	(* Get the direction of the local x-axis. *)
	METHOD GetDirectionX
	VAR_IN_OUT
		(* The local x-direction of this orientation. *)
 {attribute 'GUID' := '26B8CE0C-6327-CF56-46C9-563EF634067D'}
				localX : TangentXY;
	END_VAR
END_METHOD


	(* Get the direction of the local y-axis. *)
	METHOD GetDirectionY
	VAR_IN_OUT
		(* The local y-direction of this orientation. *)
 {attribute 'GUID' := '26B8CE0C-6327-CF56-46C9-563EF634067D'}
				localY : TangentXY;
	END_VAR
END_METHOD


	(* Invert this position. *)
	METHOD Invert
END_METHOD


	(* Multiply an orientation to this orientation. *)
	METHOD ConcatenateWith
	VAR_IN_OUT
		(* Orientation to concatenate with. *)
 {attribute 'GUID' := 'ECEACC25-61F8-C229-5DF2-DD8132935CEE'}
				orientation2D : Orientation2D;
	END_VAR
END_METHOD


	(* Turn the orientation. *)
	METHOD TurnByC
	VAR_INPUT
		(* Rotation angle to turn by in degrees [°]. *)
		angle : LREAL;
	END_VAR
END_METHOD


	(* Rotate a PositionXY according to this orientation. *)
	METHOD Transform
	VAR_IN_OUT
		(* The orientation to multipy by. *)
 {attribute 'GUID' := '96F2C7F9-077A-C570-41B3-040B08209702'}
				positionXY : PositionXY;
	END_VAR
END_METHOD


	PROPERTY angle : LREAL
SET
END_SET
GET
END_GET
END_PROPERTY

END_FUNCTION_BLOCK

// POUs/Spatial/Functions/ConcatenateABC

	{attribute 'TcIecLibraryType'}
	{attribute 'external_name' := 'ConcatenateABC_GUID_186C30DE_4777_CF4B_4981_F8D310866484'}
	(* Concatenate two instances of Orientation3D. *)
	FUNCTION ConcatenateABC : BOOL
	VAR_IN_OUT
		rotation0	:	Orientation3D;	(* 1st input orientation of the concatenation. *)
		rotation1	:	Orientation3D;	(* 2nd input orientation of the concatenation. *)
		concatenation	:	Orientation3D;	(* The concatenation of the two input instances. *)
	END_VAR

END_FUNCTION

// POUs/Spatial/Positions/Orientation3D

	{attribute 'c++_compatible'}
	{attribute 'external_name' := 'Orientation3D_GUID_88260D10_4258_CB4B_4E9C_4A364CDA3C22'}
	{attribute 'TcIecLibraryType'}
	{attribute 'no_explicit_call' :='do not call this POU directly'}
	{attribute 'no_assign'}
	(* 3D orientation. All angles in degrees [°]. *)
	FUNCTION_BLOCK Orientation3D
	VAR
		(* Rotation around the 1st local axis in degrees [°]. *)
		p0 : LREAL;
		(* Rotation around 2nd local axis in degrees [°]. *)
		p1 : LREAL;
		(* Rotation around 3rd local axis in degrees [°]. *)
		p2 : LREAL;
		(* Defines the rotation order (rotate around local axes from left to right) *)
		 {attribute 'GUID' := 'BF8BCC1E-925E-4A57-801C-CC42AFDDA86D'}
		coordinates : E_RotationCoordinates := E_RotationCoordinates.CBA;
		 {attribute 'hide'}
		_reserved1 : ARRAY [1..84] OF USINT;
	END_VAR


	(* Internal method *)
	{attribute 'hide'}
	METHOD FB_init : BOOL
	VAR_INPUT
		(*  if TRUE, the retain variables are initialized (warm start / cold start) *)
		bInitRetains : BOOL;
		(*  if TRUE, the instance afterwards gets moved into the copy code (online change) *)
		bInCopyCode : BOOL;
	END_VAR
END_METHOD


	(* Internal method *)
	{attribute 'hide'}
	METHOD FB_exit : BOOL
	VAR_INPUT
		(*  if TRUE, the exit method is called for exiting an instance that is copied afterwards (online change). *)
		bInCopyCode : BOOL;
	END_VAR
END_METHOD


	(* Set the components of this vector to '0.0'. *)
	METHOD SetZero
END_METHOD


	(* Set the components of this position. *)
	METHOD SetValues
	VAR_IN_OUT
		(* The position values to set. *)
 {attribute 'GUID' := '88260D10-4258-CB4B-4E9C-4A364CDA3C22'}
				orientation3D : Orientation3D;
	END_VAR
END_METHOD


	(* Set the coordinates of the orientation. *)
	METHOD SetValuesABC
	VAR_INPUT
		(* 1st rotation angle in degrees [°]. *)
		phi0 : LREAL;
		(* 2nd rotation angle in degrees [°]. *)
		phi1 : LREAL;
		(* 3rd rotation angle in degrees [°]. *)
		phi2 : LREAL;
	END_VAR
END_METHOD


	(* Set the coordinates of the orientation. *)
	METHOD SetValuesACB
	VAR_INPUT
		(* 1st rotation angle in degrees [°]. *)
		phi0 : LREAL;
		(* 2nd rotation angle in degrees [°]. *)
		phi1 : LREAL;
		(* 3rd rotation angle in degrees [°]. *)
		phi2 : LREAL;
	END_VAR
END_METHOD


	(* Set the coordinates of the orientation. *)
	METHOD SetValuesBCA
	VAR_INPUT
		(* 1st rotation angle in degrees [°]. *)
		phi0 : LREAL;
		(* 2nd rotation angle in degrees [°]. *)
		phi1 : LREAL;
		(* 3rd rotation angle in degrees [°]. *)
		phi2 : LREAL;
	END_VAR
END_METHOD


	(* Set the coordinates of the orientation. *)
	METHOD SetValuesBAC
	VAR_INPUT
		(* 1st rotation angle in degrees [°]. *)
		phi0 : LREAL;
		(* 2nd rotation angle in degrees [°]. *)
		phi1 : LREAL;
		(* 3rd rotation angle in degrees [°]. *)
		phi2 : LREAL;
	END_VAR
END_METHOD


	(* Set the coordinates of the orientation. *)
	METHOD SetValuesCAB
	VAR_INPUT
		(* 1st rotation angle in degrees [°]. *)
		phi0 : LREAL;
		(* 2nd rotation angle in degrees [°]. *)
		phi1 : LREAL;
		(* 3rd rotation angle in degrees [°]. *)
		phi2 : LREAL;
	END_VAR
END_METHOD


	(* Set the coordinates of the orientation. *)
	METHOD SetValuesCBA
	VAR_INPUT
		(* 1st rotation angle in degrees [°]. *)
		phi0 : LREAL;
		(* 2nd rotation angle in degrees [°]. *)
		phi1 : LREAL;
		(* 3rd rotation angle in degrees [°]. *)
		phi2 : LREAL;
	END_VAR
END_METHOD


	(* Set the coordinates of the orientation. *)
	METHOD SetValuesABA
	VAR_INPUT
		(* 1st rotation angle in degrees [°]. *)
		phi0 : LREAL;
		(* 2nd rotation angle in degrees [°]. *)
		phi1 : LREAL;
		(* 3rd rotation angle in degrees [°]. *)
		phi2 : LREAL;
	END_VAR
END_METHOD


	(* Set the coordinates of the orientation. *)
	METHOD SetValuesACA
	VAR_INPUT
		(* 1st rotation angle in degrees [°]. *)
		phi0 : LREAL;
		(* 2nd rotation angle in degrees [°]. *)
		phi1 : LREAL;
		(* 3rd rotation angle in degrees [°]. *)
		phi2 : LREAL;
	END_VAR
END_METHOD


	(* Set the coordinates of the orientation. *)
	METHOD SetValuesBCB
	VAR_INPUT
		(* 1st rotation angle in degrees [°]. *)
		phi0 : LREAL;
		(* 2nd rotation angle in degrees [°]. *)
		phi1 : LREAL;
		(* 3rd rotation angle in degrees [°]. *)
		phi2 : LREAL;
	END_VAR
END_METHOD


	(* Set the coordinates of the orientation. *)
	METHOD SetValuesBAB
	VAR_INPUT
		(* 1st rotation angle in degrees [°]. *)
		phi0 : LREAL;
		(* 2nd rotation angle in degrees [°]. *)
		phi1 : LREAL;
		(* 3rd rotation angle in degrees [°]. *)
		phi2 : LREAL;
	END_VAR
END_METHOD


	(* Set the coordinates of the orientation. *)
	METHOD SetValuesCAC
	VAR_INPUT
		(* 1st rotation angle in degrees [°]. *)
		phi0 : LREAL;
		(* 2nd rotation angle in degrees [°]. *)
		phi1 : LREAL;
		(* 3rd rotation angle in degrees [°]. *)
		phi2 : LREAL;
	END_VAR
END_METHOD


	(* Set the coordinates of the orientation. *)
	METHOD SetValuesCBC
	VAR_INPUT
		(* 1st rotation angle in degrees [°]. *)
		phi0 : LREAL;
		(* 2nd rotation angle in degrees [°]. *)
		phi1 : LREAL;
		(* 3rd rotation angle in degrees [°]. *)
		phi2 : LREAL;
	END_VAR
END_METHOD


	(* Get the direction of the local x-axis. *)
	METHOD GetDirectionX
	VAR_IN_OUT
		(* The local x-direction of this orientation. *)
 {attribute 'GUID' := 'F5C610D1-97C6-C19E-7CED-E3534BCC46DA'}
				localX : Tangent3D;
	END_VAR
END_METHOD


	(* Get the direction of the local y-axis. *)
	METHOD GetDirectionY
	VAR_IN_OUT
		(* The local y-direction of this orientation. *)
 {attribute 'GUID' := 'F5C610D1-97C6-C19E-7CED-E3534BCC46DA'}
				localY : Tangent3D;
	END_VAR
END_METHOD


	(* Get the direction of the local z-axis. *)
	METHOD GetDirectionZ
	VAR_IN_OUT
		(* The local z-direction of this orientation. *)
 {attribute 'GUID' := 'F5C610D1-97C6-C19E-7CED-E3534BCC46DA'}
				localZ : Tangent3D;
	END_VAR
END_METHOD


	(* Invert this position. *)
	METHOD Invert
END_METHOD


	(* Multiply an orientation to this orientation. *)
	METHOD ConcatenateWith
	VAR_IN_OUT
		(* Orientation to concatenate with. *)
 {attribute 'GUID' := '88260D10-4258-CB4B-4E9C-4A364CDA3C22'}
				orientation : Orientation3D;
	END_VAR
END_METHOD


	(* Rotate around an arbitrary local axis. The turn angle is given by the length of the axis. *)
	METHOD TurnBy
	VAR_IN_OUT
		(* The axis of rotation. Its length represents the angle of rotation in degrees [°]. *)
 {attribute 'GUID' := '079EE0EF-BB9A-C328-4691-0C1D9775AB9B'}
				axis : TangentABC;
	END_VAR
END_METHOD


	(* Rotation around the local x-axis. *)
	METHOD TurnByA
	VAR_INPUT
		(* The angle to rotate by in degrees [°]. *)
		da : LREAL;
	END_VAR
END_METHOD


	(* Rotation around the local y-axis. *)
	METHOD TurnByB
	VAR_INPUT
		(* The angle to rotate by in degrees [°]. *)
		db : LREAL;
	END_VAR
END_METHOD


	(* Rotation around the local z-axis. *)
	METHOD TurnByC
	VAR_INPUT
		(* The angle to rotate by in degrees [°]. *)
		dc : LREAL;
	END_VAR
END_METHOD


	(* Rotate a Position3D according to this orientation. *)
	METHOD Transform
	VAR_IN_OUT
		(* Position to transform. *)
 {attribute 'GUID' := '2AB870EB-68E4-CB90-6B70-58195CE52F48'}
				position3D : Position3D;
	END_VAR
END_METHOD


	PROPERTY phi0 : LREAL
SET
END_SET
GET
END_GET
END_PROPERTY


	PROPERTY phi1 : LREAL
SET
END_SET
GET
END_GET
END_PROPERTY


	PROPERTY phi2 : LREAL
SET
END_SET
GET
END_GET
END_PROPERTY


	PROPERTY convention : E_RotationCoordinates
SET
END_SET
GET
END_GET
END_PROPERTY

END_FUNCTION_BLOCK

// POUs/Spatial/Functions/ConcatenateXYC

	{attribute 'TcIecLibraryType'}
	{attribute 'external_name' := 'ConcatenateXYC_GUID_3FF36687_1D56_CFED_49BA_E16821D33A61'}
	(* Concatenate two instances of PositionXYC. *)
	FUNCTION ConcatenateXYC : BOOL
	VAR_IN_OUT
		position0	:	PositionXYC;	(* 1st input position of the concatenation. *)
		position1	:	PositionXYC;	(* 2nd input position of the concatenation. *)
		concatenation	:	PositionXYC;	(* The concatenation of the two input instances. *)
	END_VAR

END_FUNCTION

// POUs/Spatial/Functions/AddXY

	{attribute 'TcIecLibraryType'}
	{attribute 'external_name' := 'AddXY_GUID_9AF6CBF8_E886_C1CE_7D79_B6347AC56EDE'}
	(* Add two instances of TangentXY. *)
	FUNCTION AddXY : BOOL
	VAR_IN_OUT
		tangent0	:	TangentXY;	(* 1st input tangent vector. *)
		tangent1	:	TangentXY;	(* 2nd input tangent vector. *)
		sumTangent	:	TangentXY;	(* Sum of the two tangent vectors. *)
	END_VAR

END_FUNCTION

// POUs/Spatial/Functions/SubtractXY

	{attribute 'TcIecLibraryType'}
	{attribute 'external_name' := 'SubtractXY_GUID_4B4AC809_E392_C314_4C45_4DF45CDC0C29'}
	(* Subtract two instances of TangentXY. *)
	FUNCTION SubtractXY : BOOL
	VAR_IN_OUT
		tangent0	:	TangentXY;	(* 1st input tangent vector. *)
		tangent1	:	TangentXY;	(* 2nd input tangent vector. *)
		difference	:	TangentXY;	(* Difference of the two tangent vectors. *)
	END_VAR

END_FUNCTION

// POUs/Spatial/Functions/MultiplyXY

	{attribute 'TcIecLibraryType'}
	{attribute 'external_name' := 'MultiplyXY_GUID_85E13E1D_F467_C3B1_4BCC_CCAD43989479'}
	(* Multiply a TangentXY by a scalar and return the result. *)
	FUNCTION MultiplyXY : BOOL
	VAR_IN_OUT
		tangent	:	TangentXY;	(* Tangent vector to multiply. *)
	END_VAR
	VAR_INPUT
		scalar	:	LREAL;	(* Scalar value to multiply with. *)
	END_VAR
	VAR_IN_OUT
		scaled	:	TangentXY;	(* Scaled input tangent vector. *)
	END_VAR

END_FUNCTION

// POUs/Spatial/Functions/ScalarXY

	{attribute 'TcIecLibraryType'}
	{attribute 'external_name' := 'ScalarXY_GUID_93FCFE61_1A57_C568_4366_FB966945F7BE'}
	(* Compute the scalar product of two instance of TangentXY. *)
	FUNCTION ScalarXY : LREAL
	VAR_IN_OUT
		tangent0	:	TangentXY;	(* 1st input tangent vector. *)
		tangent1	:	TangentXY;	(* 2nd input tangent vector. *)
	END_VAR

END_FUNCTION

// POUs/Spatial/Functions/Add3D

	{attribute 'TcIecLibraryType'}
	{attribute 'external_name' := 'Add3D_GUID_59367F1B_539F_CD33_6456_DF2799B8BB05'}
	(* Add two instances of Tangent3D. *)
	FUNCTION Add3D : BOOL
	VAR_IN_OUT
		tangent0	:	Tangent3D;	(* 1st input tangent vector. *)
		tangent1	:	Tangent3D;	(* 2nd input tangent vector. *)
		sumTangent	:	Tangent3D;	(* Sum of the two tangent vectors. *)
	END_VAR

END_FUNCTION

// POUs/Spatial/Functions/Subtract3D

	{attribute 'TcIecLibraryType'}
	{attribute 'external_name' := 'Subtract3D_GUID_4490D74F_E885_C89D_4A9C_8B24E18A51D7'}
	(* Subtract two instances of Tangent3D. *)
	FUNCTION Subtract3D : BOOL
	VAR_IN_OUT
		tangent0	:	Tangent3D;	(* 1st input tangent vector. *)
		tangent1	:	Tangent3D;	(* 2nd input tangent vector. *)
		difference	:	Tangent3D;	(* Difference of the two tangent vectors. *)
	END_VAR

END_FUNCTION

// POUs/Spatial/Functions/Multiply3D

	{attribute 'TcIecLibraryType'}
	{attribute 'external_name' := 'Multiply3D_GUID_383573DC_E2EF_CCC1_44E2_29017F46A5D5'}
	(* Multiply a Tangent3D by a scalar. *)
	FUNCTION Multiply3D : BOOL
	VAR_IN_OUT
		tangent	:	Tangent3D;	(* Tangent vector to multiply. *)
	END_VAR
	VAR_INPUT
		scalar	:	LREAL;	(* Scalar value to multiply with. *)
	END_VAR
	VAR_IN_OUT
		scaled	:	Tangent3D;	(* Scaled input tangent vector. *)
	END_VAR

END_FUNCTION

// POUs/Spatial/Functions/Scalar3D

	{attribute 'TcIecLibraryType'}
	{attribute 'external_name' := 'Scalar3D_GUID_CDD5D329_BF8D_CFD8_59AB_AE11960F9E3D'}
	(* Compute the scalar product of two instances of Tangent3D. *)
	FUNCTION Scalar3D : LREAL
	VAR_IN_OUT
		tangent0	:	Tangent3D;	(* 1st input tangent vector. *)
		tangent1	:	Tangent3D;	(* 2nd input tangent vector. *)
	END_VAR

END_FUNCTION

// POUs/Spatial/Functions/Cross3D

	{attribute 'TcIecLibraryType'}
	{attribute 'external_name' := 'Cross3D_GUID_18FD21AE_F556_CC15_6188_E6099864EA00'}
	(* Compute the cross product of two instances of Tangent3D. *)
	FUNCTION Cross3D : BOOL
	VAR_IN_OUT
		tangent0	:	Tangent3D;	(* 1st input tangent vector. *)
		tangent1	:	Tangent3D;	(* 2nd input tangent vector. *)
		crossProduct	:	Tangent3D;	(* The resulting cross product. *)
	END_VAR

END_FUNCTION

// POUs/Spatial/Functions/AddABC

	{attribute 'TcIecLibraryType'}
	{attribute 'external_name' := 'AddABC_GUID_C8FBE575_5501_C20B_7B10_541D2B8D8FAB'}
	(* Add two instances of TangentABC. *)
	FUNCTION AddABC : BOOL
	VAR_IN_OUT
		tangent0	:	TangentABC;	(* 1st input tangent vector. *)
		tangent1	:	TangentABC;	(* 2nd input tangent vector. *)
		sumTangent	:	TangentABC;	(* Sum of the two tangent vectors. *)
	END_VAR

END_FUNCTION

// POUs/Spatial/Functions/SubtractABC

	{attribute 'TcIecLibraryType'}
	{attribute 'external_name' := 'SubtractABC_GUID_75447D74_7EE7_C0D8_4EE5_65C72445BC2E'}
	(* Subtract two instances of TangentABC. *)
	FUNCTION SubtractABC : BOOL
	VAR_IN_OUT
		tangent0	:	TangentABC;	(* 1st input tangent vector. *)
		tangent1	:	TangentABC;	(* 2nd input tangent vector. *)
		difference	:	TangentABC;	(* Difference of the two tangent vectors. *)
	END_VAR

END_FUNCTION

// POUs/Spatial/Functions/MultiplyABC

	{attribute 'TcIecLibraryType'}
	{attribute 'external_name' := 'MultiplyABC_GUID_B5567C7B_8039_CF9D_597F_679077B14500'}
	(* Multiply a TangentABC by a scalar. *)
	FUNCTION MultiplyABC : BOOL
	VAR_IN_OUT
		tangent	:	TangentABC;	(* Tangent vector to multiply. *)
	END_VAR
	VAR_INPUT
		scalar	:	LREAL;	(* Scalar value to multiply with. *)
	END_VAR
	VAR_IN_OUT
		scaled	:	TangentABC;	(* Scaled input tangent vector. *)
	END_VAR

END_FUNCTION

// POUs/Spatial/Functions/AddXYC

	{attribute 'TcIecLibraryType'}
	{attribute 'external_name' := 'AddXYC_GUID_6597480E_11BA_C407_44FC_28CB30711289'}
	(* Add two instances of TangentXYC. *)
	FUNCTION AddXYC : BOOL
	VAR_IN_OUT
		tangent0	:	TangentXYC;	(* 1st input tangent vector. *)
		tangent1	:	TangentXYC;	(* 2nd input tangent vector. *)
		sumTangent	:	TangentXYC;	(* Sum of the two tangent vectors. *)
	END_VAR

END_FUNCTION

// POUs/Spatial/Functions/SubtractXYC

	{attribute 'TcIecLibraryType'}
	{attribute 'external_name' := 'SubtractXYC_GUID_A66A1E91_4274_CA5D_7BE9_ABF8824078CE'}
	(* Subtract two instances of TangentXYC. *)
	FUNCTION SubtractXYC : BOOL
	VAR_IN_OUT
		tangent0	:	TangentXYC;	(* 1st input tangent vector. *)
		tangent1	:	TangentXYC;	(* 2nd input tangent vector. *)
		difference	:	TangentXYC;	(* Difference of the two tangent vectors. *)
	END_VAR

END_FUNCTION

// POUs/Spatial/Functions/MultiplyXYC

	{attribute 'TcIecLibraryType'}
	{attribute 'external_name' := 'MultiplyXYC_GUID_10B08A83_42B7_C12E_7EDD_506DEB6C7E94'}
	(* Multiply a TangentXYC by a scalar. *)
	FUNCTION MultiplyXYC : BOOL
	VAR_IN_OUT
		tangent	:	TangentXYC;	(* Tangent vector to multiply. *)
	END_VAR
	VAR_INPUT
		scalar	:	LREAL;	(* Scalar value to multiply with. *)
	END_VAR
	VAR_IN_OUT
		scaled	:	TangentXYC;	(* Scaled input tangent vector. *)
	END_VAR

END_FUNCTION

// POUs/Spatial/Functions/Add6D

	{attribute 'TcIecLibraryType'}
	{attribute 'external_name' := 'Add6D_GUID_70971E3D_141C_C82B_491A_28750F021F76'}
	(* Add two instances of Tangent6D. *)
	FUNCTION Add6D : BOOL
	VAR_IN_OUT
		tangent0	:	Tangent6D;	(* 1st input tangent vector. *)
		tangent1	:	Tangent6D;	(* 2nd input tangent vector. *)
		sumTangent	:	Tangent6D;	(* Sum of the two tangent vectors. *)
	END_VAR

END_FUNCTION

// POUs/Spatial/Functions/Subtract6D

	{attribute 'TcIecLibraryType'}
	{attribute 'external_name' := 'Subtract6D_GUID_850464F7_0919_C7C4_6C69_D5D4CC7F433D'}
	(* Subtract two instances of Tangent6D. *)
	FUNCTION Subtract6D : BOOL
	VAR_IN_OUT
		tangent0	:	Tangent6D;	(* 1st input tangent vector. *)
		tangent1	:	Tangent6D;	(* 2nd input tangent vector. *)
		difference	:	Tangent6D;	(* Difference of the two tangent vectors. *)
	END_VAR

END_FUNCTION

// POUs/Spatial/Functions/Multiply6D

	{attribute 'TcIecLibraryType'}
	{attribute 'external_name' := 'Multiply6D_GUID_91590C66_6BA7_C429_76E4_214A1B0FF139'}
	(* Multiply a Tangent6D by a scalar. *)
	FUNCTION Multiply6D : BOOL
	VAR_IN_OUT
		tangent	:	Tangent6D;	(* Tangent vector to multiply. *)
	END_VAR
	VAR_INPUT
		scalar	:	LREAL;	(* Scalar value to multiply with. *)
	END_VAR
	VAR_IN_OUT
		scaled	:	Tangent6D;	(* Scaled input tangent vector. *)
	END_VAR

END_FUNCTION

// POUs/Spatial/Functions/ConvertToCartesian2D

	{attribute 'TcIecLibraryType'}
	{attribute 'external_name' := 'ConvertToCartesian2D_GUID_1DE05828_63AC_CD5B_493C_397BF5B8F2DA'}
	(* Convert local XYC-dynamic properties to global XY ones. *)
	FUNCTION ConvertToCartesian2D : BOOL
	VAR_IN_OUT
		position	:	PositionXYC;	(* The position hosting the local dynamic state. *)
		velocity	:	TangentXYC;	(* The local velocity vector. *)
		acceleration	:	TangentXYC;	(* The local acceleration vector. *)
		velocity_XY	:	TangentXY;	(* The resulting global Cartesian velocity. *)
		acceleration_XY	:	TangentXY;	(* The resulting global Cartesian acceleration. *)
	END_VAR

END_FUNCTION

// POUs/Shapes/Geometry2D/Container2D

	{attribute 'c++_compatible'}
	{attribute 'external_name' := 'Container2D_GUID_315B01A2_C609_C244_71C6_4F8CF4BA2CAC'}
	{attribute 'TcIecLibraryType'}
	{attribute 'no_explicit_call' :='do not call this POU directly'}
	{attribute 'no_assign'}
	FUNCTION_BLOCK Container2D EXTENDS Geometry2D


	(* Internal method *)
	METHOD FB_init : BOOL
	VAR_INPUT
		(*  if TRUE, the retain variables are initialized (warm start / cold start) *)
		bInitRetains : BOOL;
		(*  if TRUE, the instance afterwards gets moved into the copy code (online change) *)
		bInCopyCode : BOOL;
	END_VAR
END_METHOD


	(* Internal method *)
	{attribute 'hide'}
	METHOD FB_exit : BOOL
	VAR_INPUT
		(*  if TRUE, the exit method is called for exiting an instance that is copied afterwards (online change). *)
		bInCopyCode : BOOL;
	END_VAR
END_METHOD


	(* Add a geometry to the container. *)
	METHOD AddElement : UDINT
	VAR_IN_OUT
		(* The geometry to add. *)
 {attribute 'GUID' := 'AD3CB6DF-15CC-CB02-52B0-F7F4EE14B341'}
				inputObject : Geometry2D;
	END_VAR
END_METHOD


	(* Remove a specified geometry from the container. *)
	METHOD RemoveElement
	VAR_INPUT
		(* ID of the geometry to remove. *)
		id : UDINT;
	END_VAR
END_METHOD


	(* Remove all geometries from the container. *)
	METHOD Clear
END_METHOD


	(* Get the number of geometry elements in container. *)
	METHOD GetCount : UDINT
END_METHOD


	(* Get the combined boundary of all hosted 2D-geometries. *)
	METHOD GetBoundary
	VAR_IN_OUT
		(* The combined boundary.. *)
 {attribute 'GUID' := '315B01A2-C609-C244-71C6-4F8CF4BA2CAC'}
				boundary : Container2D;
	END_VAR
END_METHOD

END_FUNCTION_BLOCK

// POUs/Shapes/Geometry2D/Extrude2D

	{attribute 'c++_compatible'}
	{attribute 'external_name' := 'Extrude2D_GUID_A7398709_3D7C_C1FD_7FCC_D371605A7865'}
	{attribute 'TcIecLibraryType'}
	{attribute 'no_explicit_call' :='do not call this POU directly'}
	{attribute 'no_assign'}
	FUNCTION_BLOCK Extrude2D EXTENDS Geometry2D


	(* Internal method *)
	METHOD FB_init : BOOL
	VAR_INPUT
		(*  if TRUE, the retain variables are initialized (warm start / cold start) *)
		bInitRetains : BOOL;
		(*  if TRUE, the instance afterwards gets moved into the copy code (online change) *)
		bInCopyCode : BOOL;
	END_VAR
END_METHOD


	(* Internal method *)
	{attribute 'hide'}
	METHOD FB_exit : BOOL
	VAR_INPUT
		(*  if TRUE, the exit method is called for exiting an instance that is copied afterwards (online change). *)
		bInCopyCode : BOOL;
	END_VAR
END_METHOD


	(* Define the extrusion geometry by a path and the corners to extrude. *)
	METHOD ExtrudeAlong
	VAR_IN_OUT
		(* The path to extrude along. *)
 {attribute 'GUID' := '044C9999-A9FC-C11F-572C-C4386A916232'}
				path : PathXYC;
	END_VAR
	VAR_INPUT
		(* 1st distance from the path to extrude. *)
		dy0 : LREAL;
		(* 2nd distance from the path to extrude. *)
		dy1 : LREAL;
		(* Number of steps to employ along the path. *)
		extrusionSteps : UDINT;
	END_VAR
END_METHOD


	(* Check whether this extrusion geometry is valid. *)
	METHOD IsValid : BOOL
END_METHOD

END_FUNCTION_BLOCK

// POUs/Paths/Components/PathXYC

	{attribute 'c++_compatible'}
	{attribute 'external_name' := 'PathXYC_GUID_044C9999_A9FC_C11F_572C_C4386A916232'}
	{attribute 'TcIecLibraryType'}
	{attribute 'no_explicit_call' :='do not call this POU directly'}
	{attribute 'no_assign'}
	(* A path in the xy-plane with an additional orientation at every path position. *)
	FUNCTION_BLOCK PathXYC EXTENDS IPlcPath2D


	(* Internal method *)
	{attribute 'hide'}
	METHOD FB_init : BOOL
	VAR_INPUT
		(*  if TRUE, the retain variables are initialized (warm start / cold start) *)
		bInitRetains : BOOL;
		(*  if TRUE, the instance afterwards gets moved into the copy code (online change) *)
		bInCopyCode : BOOL;
	END_VAR
END_METHOD


	(* Internal method *)
	{attribute 'hide'}
	METHOD FB_exit : BOOL
	VAR_INPUT
		(*  if TRUE, the exit method is called for exiting an instance that is copied afterwards (online change). *)
		bInCopyCode : BOOL;
	END_VAR
END_METHOD


	(* Append a smooth transition from the current end of the path
            to the specified position. *)
	METHOD AppendPosition
	VAR_IN_OUT
		(* The position to append. *)
 {attribute 'GUID' := '13C87E44-6A98-CD36-549C-47FF86B172B0'}
				position : PositionXYC;
	END_VAR
END_METHOD


	(* Append a smooth transition from the current end of the path
            to the specified position. *)
	METHOD AppendPositionXYC
	VAR_INPUT
		(* x-component of the position to append. *)
		x : LREAL;
		(* y-component of the position to append. *)
		y : LREAL;
		(* c-component of the position to append in degrees [°]. *)
		c : LREAL;
	END_VAR
END_METHOD


	(* Append a line to this path. *)
	METHOD AppendLine
	VAR_IN_OUT
		(* Start position of the line. *)
 {attribute 'GUID' := '13C87E44-6A98-CD36-549C-47FF86B172B0'}
				startPos : PositionXYC;
		(* End position of the line. *)
 {attribute 'GUID' := '13C87E44-6A98-CD36-549C-47FF86B172B0'}
				endPos : PositionXYC;
	END_VAR
END_METHOD


	(* Append a circle to this path. *)
	METHOD AppendCircle
	VAR_IN_OUT
		(* Start position of the circle. *)
 {attribute 'GUID' := '13C87E44-6A98-CD36-549C-47FF86B172B0'}
				startPos : PositionXYC;
		(* End position of the circle. *)
 {attribute 'GUID' := '13C87E44-6A98-CD36-549C-47FF86B172B0'}
				endPos : PositionXYC;
		(* Center of the circle. *)
 {attribute 'GUID' := '96F2C7F9-077A-C570-41B3-040B08209702'}
				center : PositionXY;
	END_VAR
	VAR_INPUT
		(* Set whether the circle runs clockwise or counter-clockwise. *)
		clockwise : BOOL;
	END_VAR
END_METHOD


	(* Appends a smooth transition from the end of this path
              to the start of the other path, locking further changes of this path. *)
	METHOD EndAtPath
	VAR_IN_OUT
		(* The other path. *)
 {attribute 'GUID' := '044C9999-A9FC-C11F-572C-C4386A916232'}
				path : PathXYC;
	END_VAR
END_METHOD


	(* Appends a smooth transition from the start of this path
              to the end of the other path, locking further changes of the other path. *)
	METHOD StartFromPath
	VAR_IN_OUT
		(* The other path. *)
 {attribute 'GUID' := '044C9999-A9FC-C11F-572C-C4386A916232'}
				path : PathXYC;
	END_VAR
END_METHOD


	(* Connect start and end position.
              A smooth transition is added as long as start and end positin are not identical.
              This operation finalizes this path defintion and locks it against further modifications. *)
	METHOD CloseLoop
END_METHOD


	(* Empty all current path definitions and reset the path back to an empty state. *)
	METHOD Clear
END_METHOD


	(* Get the start position of the path. *)
	METHOD GetStartPosition
	VAR_IN_OUT
		(* The current start position of the path. *)
 {attribute 'GUID' := '13C87E44-6A98-CD36-549C-47FF86B172B0'}
				startPosition : PositionXYC;
	END_VAR
END_METHOD


	(* Get the end position of the segment. *)
	METHOD GetEndPosition
	VAR_IN_OUT
		(* The current end position of the segment. *)
 {attribute 'GUID' := '13C87E44-6A98-CD36-549C-47FF86B172B0'}
				endPosition : PositionXYC;
	END_VAR
END_METHOD


	(* Get a position on the path at a specific arclength value. *)
	METHOD GetPositionAt
	VAR_INPUT
		(* Arc length value where the position is evaluated. *)
		arcLength : LREAL;
	END_VAR
	VAR_IN_OUT
		(* The position at the specified arc parameter. *)
 {attribute 'GUID' := '13C87E44-6A98-CD36-549C-47FF86B172B0'}
				position : PositionXYC;
	END_VAR
END_METHOD


	(* Get the dynamic information when moving along a path
            with specific arclength value and dynamic changes. *)
	METHOD GetStateAt
	VAR_INPUT
		(* Arc length value where the position is evaluated. *)
		arcLength : LREAL;
		(* Velocity of the arc length parameter. *)
		arcVelocity : LREAL;
		(* Acceleration of the arc length parameter. *)
		arcAcceleration : LREAL;
	END_VAR
	VAR_IN_OUT
		(* The position at the specified arc parameter. *)
 {attribute 'GUID' := '13C87E44-6A98-CD36-549C-47FF86B172B0'}
				position : PositionXYC;
		(* The velocity at the specified dynamic state. *)
 {attribute 'GUID' := 'A7123A6A-F113-C0C1-5FAB-8A846FF5D5BE'}
				velocity : TangentXYC;
		(* The acceleration at the specified dynamic state. *)
 {attribute 'GUID' := 'A7123A6A-F113-C0C1-5FAB-8A846FF5D5BE'}
				acceleration : TangentXYC;
	END_VAR
END_METHOD

END_FUNCTION_BLOCK

// POUs/Shapes/Geometry3D/Container3D

	{attribute 'c++_compatible'}
	{attribute 'external_name' := 'Container3D_GUID_9051F4D4_945A_C803_692E_DBAE727B33CC'}
	{attribute 'TcIecLibraryType'}
	{attribute 'no_explicit_call' :='do not call this POU directly'}
	{attribute 'no_assign'}
	FUNCTION_BLOCK Container3D EXTENDS Geometry3D


	(* Internal method *)
	METHOD FB_init : BOOL
	VAR_INPUT
		(*  if TRUE, the retain variables are initialized (warm start / cold start) *)
		bInitRetains : BOOL;
		(*  if TRUE, the instance afterwards gets moved into the copy code (online change) *)
		bInCopyCode : BOOL;
	END_VAR
END_METHOD


	(* Internal method *)
	{attribute 'hide'}
	METHOD FB_exit : BOOL
	VAR_INPUT
		(*  if TRUE, the exit method is called for exiting an instance that is copied afterwards (online change). *)
		bInCopyCode : BOOL;
	END_VAR
END_METHOD


	(* Add a geometry to the container. *)
	METHOD AddElement : UDINT
	VAR_IN_OUT
		(* The geometry to add. *)
 {attribute 'GUID' := '11BCDDC1-9B84-CFEE-5C12-0EC9E63800AC'}
				geometry : Geometry3D;
	END_VAR
END_METHOD


	(* Remove a specified geometry from the container. *)
	METHOD RemoveElement
	VAR_INPUT
		(* Identifier of the geometry to remove. *)
		id : UDINT;
	END_VAR
END_METHOD


	(* Remove all geometries from container. *)
	METHOD Clear
END_METHOD


	(* Get the number of geometry elements in container. *)
	METHOD GetCount : UDINT
END_METHOD

END_FUNCTION_BLOCK

// POUs/Shapes/Geometry3D/Extrude3D

	{attribute 'c++_compatible'}
	{attribute 'external_name' := 'Extrude3D_GUID_DAA935DB_549C_CB4F_6D78_E269D327B157'}
	{attribute 'TcIecLibraryType'}
	{attribute 'no_explicit_call' :='do not call this POU directly'}
	{attribute 'no_assign'}
	FUNCTION_BLOCK Extrude3D EXTENDS Geometry3D


	(* Internal method *)
	METHOD FB_init : BOOL
	VAR_INPUT
		(*  if TRUE, the retain variables are initialized (warm start / cold start) *)
		bInitRetains : BOOL;
		(*  if TRUE, the instance afterwards gets moved into the copy code (online change) *)
		bInCopyCode : BOOL;
	END_VAR
END_METHOD


	(* Internal method *)
	{attribute 'hide'}
	METHOD FB_exit : BOOL
	VAR_INPUT
		(*  if TRUE, the exit method is called for exiting an instance that is copied afterwards (online change). *)
		bInCopyCode : BOOL;
	END_VAR
END_METHOD

END_FUNCTION_BLOCK

// POUs/Paths/Components/PathXY

	{attribute 'c++_compatible'}
	{attribute 'external_name' := 'PathXY_GUID_C5A448CE_AA85_CB43_4C16_DB8A68FE6919'}
	{attribute 'TcIecLibraryType'}
	{attribute 'no_explicit_call' :='do not call this POU directly'}
	{attribute 'no_assign'}
	(* A path in the xy-plane. *)
	FUNCTION_BLOCK PathXY EXTENDS IPlcPath2D


	(* Internal method *)
	{attribute 'hide'}
	METHOD FB_init : BOOL
	VAR_INPUT
		(*  if TRUE, the retain variables are initialized (warm start / cold start) *)
		bInitRetains : BOOL;
		(*  if TRUE, the instance afterwards gets moved into the copy code (online change) *)
		bInCopyCode : BOOL;
	END_VAR
END_METHOD


	(* Internal method *)
	{attribute 'hide'}
	METHOD FB_exit : BOOL
	VAR_INPUT
		(*  if TRUE, the exit method is called for exiting an instance that is copied afterwards (online change). *)
		bInCopyCode : BOOL;
	END_VAR
END_METHOD


	(* Append a smooth transition from the current end of the path
            to the specified position. *)
	METHOD AppendPosition
	VAR_IN_OUT
		(* The position to append. *)
 {attribute 'GUID' := '96F2C7F9-077A-C570-41B3-040B08209702'}
				position : PositionXY;
	END_VAR
END_METHOD


	(* Append a smooth transition from the current end of the path
            to the specified position. *)
	METHOD AppendPositionXY
	VAR_INPUT
		(* x-component of the position to append. *)
		x : LREAL;
		(* y-component of the position to append. *)
		y : LREAL;
	END_VAR
END_METHOD


	(* Append a line to this path. *)
	METHOD AppendLine
	VAR_IN_OUT
		(* Start position of the line. *)
 {attribute 'GUID' := '96F2C7F9-077A-C570-41B3-040B08209702'}
				startPos : PositionXY;
		(* End position of the line. *)
 {attribute 'GUID' := '96F2C7F9-077A-C570-41B3-040B08209702'}
				endPos : PositionXY;
	END_VAR
END_METHOD


	(* Append a circle to this path. *)
	METHOD AppendCircle
	VAR_IN_OUT
		(* Start position of the circle. *)
 {attribute 'GUID' := '96F2C7F9-077A-C570-41B3-040B08209702'}
				startPos : PositionXY;
		(* End position of the circle. *)
 {attribute 'GUID' := '96F2C7F9-077A-C570-41B3-040B08209702'}
				endPos : PositionXY;
		(* Center of the circle. *)
 {attribute 'GUID' := '96F2C7F9-077A-C570-41B3-040B08209702'}
				center : PositionXY;
	END_VAR
	VAR_INPUT
		(* Set whether the circle runs clockwise or counter-clockwise. *)
		clockwise : BOOL;
	END_VAR
END_METHOD


	(* Get the start position of the path. *)
	METHOD GetStartPosition
	VAR_IN_OUT
		(* The current start position of the path. *)
 {attribute 'GUID' := '96F2C7F9-077A-C570-41B3-040B08209702'}
				startPosition : PositionXY;
	END_VAR
END_METHOD


	(* Get the end position of the segment. *)
	METHOD GetEndPosition
	VAR_IN_OUT
		(* The current end position of the segment. *)
 {attribute 'GUID' := '96F2C7F9-077A-C570-41B3-040B08209702'}
				endPosition : PositionXY;
	END_VAR
END_METHOD


	(* Get a position on the path at a specific arclength value. *)
	METHOD GetPositionAt
	VAR_INPUT
		(* Arc length value where the position is evaluated. *)
		arcLength : LREAL;
	END_VAR
	VAR_IN_OUT
		(* The position at the specified arc parameter. *)
 {attribute 'GUID' := '96F2C7F9-077A-C570-41B3-040B08209702'}
				position : PositionXY;
	END_VAR
END_METHOD


	(* Get the dynamic information when moving along a path
            with specific arclength value and dynamic changes. *)
	METHOD GetStateAt
	VAR_INPUT
		(* Arc length value where the position is evaluated. *)
		arcLength : LREAL;
		(* Velocity of the arc length parameter. *)
		arcVelocity : LREAL;
		(* Acceleration of the arc length parameter. *)
		arcAcceleration : LREAL;
	END_VAR
	VAR_IN_OUT
		(* The position at the specified arc parameter. *)
 {attribute 'GUID' := '96F2C7F9-077A-C570-41B3-040B08209702'}
				position : PositionXY;
		(* The velocity at the specified dynamic state. *)
 {attribute 'GUID' := '26B8CE0C-6327-CF56-46C9-563EF634067D'}
				velocity : TangentXY;
		(* The acceleration at the specified dynamic state. *)
 {attribute 'GUID' := '26B8CE0C-6327-CF56-46C9-563EF634067D'}
				acceleration : TangentXY;
	END_VAR
END_METHOD

END_FUNCTION_BLOCK

// POUs/Paths/Components/PathXYZ

	{attribute 'c++_compatible'}
	{attribute 'external_name' := 'PathXYZ_GUID_2243D2B5_C102_C5AD_6308_697554B84920'}
	{attribute 'TcIecLibraryType'}
	{attribute 'no_explicit_call' :='do not call this POU directly'}
	{attribute 'no_assign'}
	(* A path in the xy-plane with an additional orientation at every path position. *)
	FUNCTION_BLOCK PathXYZ EXTENDS IPlcPath3D


	(* Internal method *)
	{attribute 'hide'}
	METHOD FB_init : BOOL
	VAR_INPUT
		(*  if TRUE, the retain variables are initialized (warm start / cold start) *)
		bInitRetains : BOOL;
		(*  if TRUE, the instance afterwards gets moved into the copy code (online change) *)
		bInCopyCode : BOOL;
	END_VAR
END_METHOD


	(* Internal method *)
	{attribute 'hide'}
	METHOD FB_exit : BOOL
	VAR_INPUT
		(*  if TRUE, the exit method is called for exiting an instance that is copied afterwards (online change). *)
		bInCopyCode : BOOL;
	END_VAR
END_METHOD


	(* Append a smooth transition from the current end of the path
            to the specified position. *)
	METHOD AppendPosition
	VAR_IN_OUT
		(* The position to append. *)
 {attribute 'GUID' := '2AB870EB-68E4-CB90-6B70-58195CE52F48'}
				position : Position3D;
	END_VAR
END_METHOD


	(* Append a smooth transition from the current end of the path
            to the specified position. *)
	METHOD AppendPositionXYZ
	VAR_INPUT
		(* x-component of the position to append. *)
		x : LREAL;
		(* y-component of the position to append. *)
		y : LREAL;
		(* z-component of the position to append. *)
		c : LREAL;
	END_VAR
END_METHOD


	(* Append a line to this path. *)
	METHOD AppendLine
	VAR_IN_OUT
		(* Start position of the line. *)
 {attribute 'GUID' := '2AB870EB-68E4-CB90-6B70-58195CE52F48'}
				startPos : Position3D;
		(* End position of the line. *)
 {attribute 'GUID' := '2AB870EB-68E4-CB90-6B70-58195CE52F48'}
				endPos : Position3D;
	END_VAR
END_METHOD


	(* Append a smooth transition from the current end of the path
            to the specified position. *)
	METHOD AppendLineXYZ
	VAR_INPUT
		(* x-component of the start position. *)
		x0 : LREAL;
		(* y-component of the start position. *)
		y0 : LREAL;
		(* z-component of the start position. *)
		z0 : LREAL;
		(* x-component of the end position. *)
		x1 : LREAL;
		(* y-component of the end position. *)
		y1 : LREAL;
		(* z-component of the end position. *)
		z1 : LREAL;
	END_VAR
END_METHOD


	(* Append a circle to this path. *)
	METHOD AppendCircle
	VAR_IN_OUT
		(* Start position of the circle. *)
 {attribute 'GUID' := '2AB870EB-68E4-CB90-6B70-58195CE52F48'}
				startPos : Position3D;
		(* End position of the circle. *)
 {attribute 'GUID' := '2AB870EB-68E4-CB90-6B70-58195CE52F48'}
				endPos : Position3D;
		(* Center of the circle. *)
 {attribute 'GUID' := '96F2C7F9-077A-C570-41B3-040B08209702'}
				center : PositionXY;
	END_VAR
	VAR_INPUT
		(* Set whether the circle runs clockwise or counter-clockwise. *)
		clockwise : BOOL;
	END_VAR
END_METHOD


	(* Append a smooth transition from the current end of the path
            to the specified position with tangent. *)
	METHOD AppendPositionTangent
	VAR_IN_OUT
		(* The position to append. *)
 {attribute 'GUID' := '2AB870EB-68E4-CB90-6B70-58195CE52F48'}
				position : Position3D;
		(* The tangent to append *)
 {attribute 'GUID' := 'F5C610D1-97C6-C19E-7CED-E3534BCC46DA'}
				tangent : Tangent3D;
	END_VAR
END_METHOD


	(* Get the start position of the path. *)
	METHOD GetStartPosition
	VAR_IN_OUT
		(* The current start position of the path. *)
 {attribute 'GUID' := '2AB870EB-68E4-CB90-6B70-58195CE52F48'}
				startPosition : Position3D;
	END_VAR
END_METHOD


	(* Get the end position of the segment. *)
	METHOD GetEndPosition
	VAR_IN_OUT
		(* The current end position of the segment. *)
 {attribute 'GUID' := '2AB870EB-68E4-CB90-6B70-58195CE52F48'}
				endPosition : Position3D;
	END_VAR
END_METHOD


	(* Get a position on the path at a specific arclength value. *)
	METHOD GetPositionAt
	VAR_INPUT
		(* Arc length value where the position is evaluated. *)
		arcLength : LREAL;
	END_VAR
	VAR_IN_OUT
		(* The position at the specified arc parameter. *)
 {attribute 'GUID' := '2AB870EB-68E4-CB90-6B70-58195CE52F48'}
				position : Position3D;
	END_VAR
END_METHOD


	(* Get the dynamic information when moving along a path
            with specific arclength value and dynamic changes. *)
	METHOD GetStateAt
	VAR_INPUT
		(* Arc length value where the position is evaluated. *)
		arcLength : LREAL;
		(* Velocity of the arc length parameter. *)
		arcVelocity : LREAL;
		(* Acceleration of the arc length parameter. *)
		arcAcceleration : LREAL;
	END_VAR
	VAR_IN_OUT
		(* The position at the specified arc parameter. *)
 {attribute 'GUID' := '13C87E44-6A98-CD36-549C-47FF86B172B0'}
				position : PositionXYC;
		(* The velocity at the specified dynamic state. *)
 {attribute 'GUID' := 'F5C610D1-97C6-C19E-7CED-E3534BCC46DA'}
				velocity : Tangent3D;
		(* The acceleration at the specified dynamic state. *)
 {attribute 'GUID' := 'F5C610D1-97C6-C19E-7CED-E3534BCC46DA'}
				acceleration : Tangent3D;
	END_VAR
END_METHOD

END_FUNCTION_BLOCK

// POUs/Shapes/Geometry2D/Functions/CheckCollision2D

	{attribute 'TcIecLibraryType'}
	{attribute 'external_name' := 'CheckCollision2D_GUID_8AFDC95F_F653_C66D_7F45_55F37338C1FA'}
	(* Check if two geometries are currently colliding. *)
	FUNCTION CheckCollision2D : BOOL
	VAR_IN_OUT
		geometry0	:	IPlcGeometry2D;	(* 1st input geometry to check for collision. *)
		geometry1	:	IPlcGeometry2D;	(* 2nd input geometry to check of collision. *)
	END_VAR

END_FUNCTION

// POUs/Shapes/Geometry2D/Functions/GetDistance2D

	{attribute 'TcIecLibraryType'}
	{attribute 'external_name' := 'GetDistance2D_GUID_B532B2A7_3728_CCF8_4B09_5BD2C6831C66'}
	(* Get the distance between two geometries. *)
	FUNCTION GetDistance2D : LREAL
	VAR_IN_OUT
		geometry0	:	IPlcGeometry2D;	(* 1st input geometry to calculate the distance of. *)
		geometry1	:	IPlcGeometry2D;	(* 2nd input geometry to calculate the distance of. *)
	END_VAR

END_FUNCTION

// POUs/Shapes/Geometry2D/Functions/GetLinkingLine2D

	{attribute 'TcIecLibraryType'}
	{attribute 'external_name' := 'GetLinkingLine2D_GUID_F3D9B298_45DE_C295_6F77_34498FAFB330'}
	(* Get the shortest path between two geometries. *)
	FUNCTION GetLinkingLine2D : BOOL
	VAR_IN_OUT
		geometry0	:	IPlcGeometry2D;	(* 1st input geometry to calculate the linking line for. *)
		geometry1	:	IPlcGeometry2D;	(* 2nd input geometry to calculate the linking line for. *)
		linkingLine	:	Segment2D;	(* Return the resulting linking line. *)
	END_VAR

END_FUNCTION

// POUs/Shapes/Geometry2D/1D/Segment2D

	{attribute 'c++_compatible'}
	{attribute 'external_name' := 'Segment2D_GUID_B0DCCAD8_7A88_CBE4_4347_DF93C8389EE1'}
	{attribute 'TcIecLibraryType'}
	{attribute 'no_explicit_call' :='do not call this POU directly'}
	{attribute 'no_assign'}
	FUNCTION_BLOCK Segment2D EXTENDS Geometry2D


	(* Internal method *)
	METHOD FB_init : BOOL
	VAR_INPUT
		(*  if TRUE, the retain variables are initialized (warm start / cold start) *)
		bInitRetains : BOOL;
		(*  if TRUE, the instance afterwards gets moved into the copy code (online change) *)
		bInCopyCode : BOOL;
	END_VAR
END_METHOD


	(* Internal method *)
	{attribute 'hide'}
	METHOD FB_exit : BOOL
	VAR_INPUT
		(*  if TRUE, the exit method is called for exiting an instance that is copied afterwards (online change). *)
		bInCopyCode : BOOL;
	END_VAR
END_METHOD


	(* Set the start position of the segment. *)
	METHOD SetStartPosition
	VAR_IN_OUT
		(* Start position of the segment to set. *)
 {attribute 'GUID' := '96F2C7F9-077A-C570-41B3-040B08209702'}
				startPos : PositionXY;
	END_VAR
END_METHOD


	(* Set the start position of the segment. *)
	METHOD SetStartPositionXY
	VAR_INPUT
		(* x-component of the start position. *)
		x : LREAL;
		(* y-component of the start position. *)
		y : LREAL;
	END_VAR
END_METHOD


	(* Set the end position of the segment. *)
	METHOD SetEndPosition
	VAR_IN_OUT
		(* End position of the segment to set. *)
 {attribute 'GUID' := '96F2C7F9-077A-C570-41B3-040B08209702'}
				endPos : PositionXY;
	END_VAR
END_METHOD


	(* Set the end position of the segment. *)
	METHOD SetEndPositionXY
	VAR_INPUT
		(* x-component of the end position. *)
		x : LREAL;
		(* y-component of the end position. *)
		y : LREAL;
	END_VAR
END_METHOD


	(* Get the x-component of the segment length in respect to the root coordinate system. *)
	METHOD Get_dX : LREAL
END_METHOD


	(* Get the y-component of the segment length in respect to the root coordinate system. *)
	METHOD Get_dY : LREAL
END_METHOD


	(* Get the length of the segment. *)
	METHOD GetLength : LREAL
END_METHOD


	(* Get the start position of the segment. *)
	METHOD GetStartPosition
	VAR_IN_OUT
		(* The current start position of the segment. *)
 {attribute 'GUID' := '96F2C7F9-077A-C570-41B3-040B08209702'}
				startPosition : PositionXY;
	END_VAR
END_METHOD


	(* Get the end position of the segment. *)
	METHOD GetEndPosition
	VAR_IN_OUT
		(* The current end position of the segment. *)
 {attribute 'GUID' := '96F2C7F9-077A-C570-41B3-040B08209702'}
				endPosition : PositionXY;
	END_VAR
END_METHOD


	(* Get the direction of the segment. *)
	METHOD GetDirection
	VAR_IN_OUT
		(* The current direction of the segment. *)
 {attribute 'GUID' := '26B8CE0C-6327-CF56-46C9-563EF634067D'}
				direction : TangentXY;
	END_VAR
END_METHOD


	(* Get a position on the segment at a specific arclength value. *)
	METHOD GetPositionAt
	VAR_INPUT
		(* Arc length value where the position is evaluated. *)
		arcLength : LREAL;
	END_VAR
	VAR_IN_OUT
		(* The position at the specified arc parameter. *)
 {attribute 'GUID' := '13C87E44-6A98-CD36-549C-47FF86B172B0'}
				position : PositionXYC;
	END_VAR
END_METHOD

END_FUNCTION_BLOCK

// POUs/Shapes/Geometry2D/1D/Line2D

	{attribute 'c++_compatible'}
	{attribute 'external_name' := 'Line2D_GUID_D12D2ADD_7B0E_C3FA_4011_AA4360740D3B'}
	{attribute 'TcIecLibraryType'}
	{attribute 'no_explicit_call' :='do not call this POU directly'}
	{attribute 'no_assign'}
	(* 2D Geometry Line *)
	FUNCTION_BLOCK Line2D EXTENDS Geometry2D


	(* Internal method *)
	METHOD FB_init : BOOL
	VAR_INPUT
		(*  if TRUE, the retain variables are initialized (warm start / cold start) *)
		bInitRetains : BOOL;
		(*  if TRUE, the instance afterwards gets moved into the copy code (online change) *)
		bInCopyCode : BOOL;
	END_VAR
END_METHOD


	(* Internal method *)
	{attribute 'hide'}
	METHOD FB_exit : BOOL
	VAR_INPUT
		(*  if TRUE, the exit method is called for exiting an instance that is copied afterwards (online change). *)
		bInCopyCode : BOOL;
	END_VAR
END_METHOD


	(* Define a line by two positions. *)
	METHOD DefineByPositions
	VAR_IN_OUT
		(* 1st position on the line to define. *)
 {attribute 'GUID' := '96F2C7F9-077A-C570-41B3-040B08209702'}
				position0 : PositionXY;
		(* 2nd position on the line to define. *)
 {attribute 'GUID' := '96F2C7F9-077A-C570-41B3-040B08209702'}
				position1 : PositionXY;
	END_VAR
END_METHOD


	(* Define a line by a position on the line and its direction. *)
	METHOD DefineByDirection
	VAR_IN_OUT
		(* Position on the line *)
 {attribute 'GUID' := '96F2C7F9-077A-C570-41B3-040B08209702'}
				position : PositionXY;
		(* Direction of the line *)
 {attribute 'GUID' := '26B8CE0C-6327-CF56-46C9-563EF634067D'}
				direction : TangentXY;
	END_VAR
END_METHOD


	(* Set the direction of the line. *)
	METHOD SetDirection
	VAR_IN_OUT
		(* The direction to set. *)
 {attribute 'GUID' := '26B8CE0C-6327-CF56-46C9-563EF634067D'}
				direction : TangentXY;
	END_VAR
END_METHOD


	(* Get the direction of the line. *)
	METHOD GetDirection
	VAR_IN_OUT
		(* The current direction of the line. *)
 {attribute 'GUID' := '26B8CE0C-6327-CF56-46C9-563EF634067D'}
				direction : TangentXY;
	END_VAR
END_METHOD


	(* Get a position on the line at a specific arclength value. *)
	METHOD GetPositionAt
	VAR_INPUT
		(* Arc length value where the position is evaluated. *)
		arcLength : LREAL;
	END_VAR
	VAR_IN_OUT
		(* The position at the specified arc parameter. *)
 {attribute 'GUID' := '13C87E44-6A98-CD36-549C-47FF86B172B0'}
				position : PositionXYC;
	END_VAR
END_METHOD

END_FUNCTION_BLOCK

// POUs/Shapes/Geometry2D/1D/Circle2D

	{attribute 'c++_compatible'}
	{attribute 'external_name' := 'Circle2D_GUID_E79B19AB_7614_C82D_719D_FDA3EE91DB40'}
	{attribute 'TcIecLibraryType'}
	{attribute 'no_explicit_call' :='do not call this POU directly'}
	{attribute 'no_assign'}
	FUNCTION_BLOCK Circle2D EXTENDS Geometry2D


	(* Internal method *)
	METHOD FB_init : BOOL
	VAR_INPUT
		(*  if TRUE, the retain variables are initialized (warm start / cold start) *)
		bInitRetains : BOOL;
		(*  if TRUE, the instance afterwards gets moved into the copy code (online change) *)
		bInCopyCode : BOOL;
	END_VAR
END_METHOD


	(* Internal method *)
	{attribute 'hide'}
	METHOD FB_exit : BOOL
	VAR_INPUT
		(*  if TRUE, the exit method is called for exiting an instance that is copied afterwards (online change). *)
		bInCopyCode : BOOL;
	END_VAR
END_METHOD


	(* Get the length of the circle. *)
	METHOD GetLength : LREAL
END_METHOD


	(* Get a position on the circle at a specific arclength value. *)
	METHOD GetPositionAt
	VAR_INPUT
		(* Arc length value where the position is evaluated. *)
		arcLength : LREAL;
	END_VAR
	VAR_IN_OUT
		(* The position at the specified arc parameter. *)
 {attribute 'GUID' := '13C87E44-6A98-CD36-549C-47FF86B172B0'}
				position : PositionXYC;
	END_VAR
END_METHOD


	PROPERTY radius : LREAL
SET
END_SET
GET
END_GET
END_PROPERTY

END_FUNCTION_BLOCK

// POUs/Shapes/Geometry2D/2D/Disc2D

	{attribute 'c++_compatible'}
	{attribute 'external_name' := 'Disc2D_GUID_1A6C6545_E8CF_C1DB_69DF_76C2EA80DE6C'}
	{attribute 'TcIecLibraryType'}
	{attribute 'no_explicit_call' :='do not call this POU directly'}
	{attribute 'no_assign'}
	FUNCTION_BLOCK Disc2D EXTENDS Geometry2D


	(* Internal method *)
	METHOD FB_init : BOOL
	VAR_INPUT
		(*  if TRUE, the retain variables are initialized (warm start / cold start) *)
		bInitRetains : BOOL;
		(*  if TRUE, the instance afterwards gets moved into the copy code (online change) *)
		bInCopyCode : BOOL;
	END_VAR
END_METHOD


	(* Internal method *)
	{attribute 'hide'}
	METHOD FB_exit : BOOL
	VAR_INPUT
		(*  if TRUE, the exit method is called for exiting an instance that is copied afterwards (online change). *)
		bInCopyCode : BOOL;
	END_VAR
END_METHOD


	(* Get the area of the disc. *)
	METHOD GetArea : LREAL
END_METHOD


	PROPERTY radius : LREAL
SET
END_SET
GET
END_GET
END_PROPERTY

END_FUNCTION_BLOCK

// POUs/Shapes/Geometry2D/2D/Rectangle2D

	{attribute 'c++_compatible'}
	{attribute 'external_name' := 'Rectangle2D_GUID_344E56D8_6CAA_CD93_7207_CDCBF767F17E'}
	{attribute 'TcIecLibraryType'}
	{attribute 'no_explicit_call' :='do not call this POU directly'}
	{attribute 'no_assign'}
	FUNCTION_BLOCK Rectangle2D EXTENDS Geometry2D


	(* Internal method *)
	METHOD FB_init : BOOL
	VAR_INPUT
		(*  if TRUE, the retain variables are initialized (warm start / cold start) *)
		bInitRetains : BOOL;
		(*  if TRUE, the instance afterwards gets moved into the copy code (online change) *)
		bInCopyCode : BOOL;
	END_VAR
END_METHOD


	(* Internal method *)
	{attribute 'hide'}
	METHOD FB_exit : BOOL
	VAR_INPUT
		(*  if TRUE, the exit method is called for exiting an instance that is copied afterwards (online change). *)
		bInCopyCode : BOOL;
	END_VAR
END_METHOD


	(* Set the dimensions of the rectangle. *)
	METHOD SetDimensions
	VAR_INPUT
		(* The width of the rectangle to set. *)
		width : LREAL;
		(* The height of the rectangle to set. *)
		height : LREAL;
	END_VAR
END_METHOD


	(* Get the area of the rectangle. *)
	METHOD GetArea : LREAL
END_METHOD


	PROPERTY width : LREAL
SET
END_SET
GET
END_GET
END_PROPERTY


	PROPERTY height : LREAL
SET
END_SET
GET
END_GET
END_PROPERTY

END_FUNCTION_BLOCK

// POUs/Shapes/Geometry3D/Functions/CheckCollision3D

	{attribute 'TcIecLibraryType'}
	{attribute 'external_name' := 'CheckCollision3D_GUID_1F78C5FB_8320_C935_6A13_9CE8E462348C'}
	(* Check if two geometries are currently colliding. *)
	FUNCTION CheckCollision3D : BOOL
	VAR_IN_OUT
		geometry0	:	IPlcGeometry3D;	(* 1st input geometry to check for collision. *)
		geometry1	:	IPlcGeometry3D;	(* 2nd input geometry to check of collision. *)
	END_VAR

END_FUNCTION

// POUs/Shapes/Geometry3D/Functions/GetDistance3D

	{attribute 'TcIecLibraryType'}
	{attribute 'external_name' := 'GetDistance3D_GUID_ECC1FBEE_14FA_CE31_4524_4CB058CE6134'}
	(* Get the distance between two geometries. *)
	FUNCTION GetDistance3D : LREAL
	VAR_IN_OUT
		geometry0	:	IPlcGeometry3D;	(* 1st input geometry to calculate the distance of. *)
		geometry1	:	IPlcGeometry3D;	(* 2nd input geometry to calculate the distance of. *)
	END_VAR

END_FUNCTION

// POUs/Shapes/Geometry3D/Functions/GetLinkingLine3D

	{attribute 'TcIecLibraryType'}
	{attribute 'external_name' := 'GetLinkingLine3D_GUID_8FFCF0E5_9435_C1E5_76E9_2526B8524AF6'}
	(* Get the shortest path between two geometries. *)
	FUNCTION GetLinkingLine3D : BOOL
	VAR_IN_OUT
		geometry0	:	IPlcGeometry3D;	(* 1st input geometry to calculate the linking line for. *)
		geometry1	:	IPlcGeometry3D;	(* 2nd input geometry to calculate the linking line for. *)
		linkingLine	:	Segment3D;	(* Return the resulting linking line. *)
	END_VAR

END_FUNCTION

// POUs/Shapes/Geometry3D/1D/Segment3D

	{attribute 'c++_compatible'}
	{attribute 'external_name' := 'Segment3D_GUID_E14243C0_9607_CC22_71A1_B077D372D570'}
	{attribute 'TcIecLibraryType'}
	{attribute 'no_explicit_call' :='do not call this POU directly'}
	{attribute 'no_assign'}
	FUNCTION_BLOCK Segment3D EXTENDS Geometry3D


	(* Internal method *)
	METHOD FB_init : BOOL
	VAR_INPUT
		(*  if TRUE, the retain variables are initialized (warm start / cold start) *)
		bInitRetains : BOOL;
		(*  if TRUE, the instance afterwards gets moved into the copy code (online change) *)
		bInCopyCode : BOOL;
	END_VAR
END_METHOD


	(* Internal method *)
	{attribute 'hide'}
	METHOD FB_exit : BOOL
	VAR_INPUT
		(*  if TRUE, the exit method is called for exiting an instance that is copied afterwards (online change). *)
		bInCopyCode : BOOL;
	END_VAR
END_METHOD


	(* Set the start position of the segment. *)
	METHOD SetStartPosition
	VAR_IN_OUT
		(* Start position of the segment to set. *)
 {attribute 'GUID' := '2AB870EB-68E4-CB90-6B70-58195CE52F48'}
				startPos : Position3D;
	END_VAR
END_METHOD


	(* Set the start position of the segment. *)
	METHOD SetStartPositionXYZ
	VAR_INPUT
		(* x-component of the start position. *)
		x : LREAL;
		(* y-component of the start position. *)
		y : LREAL;
		(* z-component of the start position. *)
		z : LREAL;
	END_VAR
END_METHOD


	(* Set the end position of the segment. *)
	METHOD SetEndPosition
	VAR_IN_OUT
		(* End position of the segment to set. *)
 {attribute 'GUID' := '2AB870EB-68E4-CB90-6B70-58195CE52F48'}
				endPos : Position3D;
	END_VAR
END_METHOD


	(* Set the end position of the segment. *)
	METHOD SetEndPositionXYZ
	VAR_INPUT
		(* x-component of the end position. *)
		x : LREAL;
		(* y-component of the end position. *)
		y : LREAL;
		(* z-component of the end position. *)
		z : LREAL;
	END_VAR
END_METHOD


	(* Get the x-component of the segment length in respect to the root coordinate system. *)
	METHOD Get_dX : LREAL
END_METHOD


	(* Get the y-component of the segment length in respect to the root coordinate system. *)
	METHOD Get_dY : LREAL
END_METHOD


	(* Get the z-component of the segment length in respect to the root coordinate system. *)
	METHOD Get_dZ : LREAL
END_METHOD


	(* Get the length of the segment. *)
	METHOD GetLength : LREAL
END_METHOD


	(* Get the start position of the segment. *)
	METHOD GetStartPosition
	VAR_IN_OUT
		(* The current start position of the segment. *)
 {attribute 'GUID' := '2AB870EB-68E4-CB90-6B70-58195CE52F48'}
				startPosition : Position3D;
	END_VAR
END_METHOD


	(* Get the end position of the segment. *)
	METHOD GetEndPosition
	VAR_IN_OUT
		(* The current end position of the segment. *)
 {attribute 'GUID' := '2AB870EB-68E4-CB90-6B70-58195CE52F48'}
				endPosition : Position3D;
	END_VAR
END_METHOD


	(* Get the direction of the segment. *)
	METHOD GetDirection
	VAR_IN_OUT
		(* The current direction of the segment. *)
 {attribute 'GUID' := 'F5C610D1-97C6-C19E-7CED-E3534BCC46DA'}
				direction : Tangent3D;
	END_VAR
END_METHOD


	(* Get a position on the segment at a specific arclength value. *)
	METHOD GetPositionAt
	VAR_INPUT
		(* Arc length value where the position is evaluated. *)
		arcLength : LREAL;
	END_VAR
	VAR_IN_OUT
		(* The position at the specified arc parameter. *)
 {attribute 'GUID' := '0AD402BA-F9BA-C1DC-7787-46186BA3F7DD'}
				position : PositionSE3;
	END_VAR
END_METHOD

END_FUNCTION_BLOCK

// POUs/Shapes/Geometry3D/Functions/CreateIntersection2D

	{attribute 'TcIecLibraryType'}
	{attribute 'external_name' := 'CreateIntersection2D_GUID_B3216808_6309_CA9D_69C7_C88EA71B2D72'}
	(* Create a collection of intersections along a plane definition. *)
	FUNCTION CreateIntersection2D : BOOL
	VAR_IN_OUT
		container3D	:	Container3D;	(* Input container to create the intersections of. *)
		planeFrame	:	PositionSE3;	(* The coordinate frame to indicate the origin of the plane. *)
		container2D	:	Container2D;	(* Return the resulting collection of intersection. *)
	END_VAR

END_FUNCTION

// POUs/Shapes/Geometry3D/1D/Line3D

	{attribute 'c++_compatible'}
	{attribute 'external_name' := 'Line3D_GUID_DC935152_29FB_CB06_6988_CFC334E21520'}
	{attribute 'TcIecLibraryType'}
	{attribute 'no_explicit_call' :='do not call this POU directly'}
	{attribute 'no_assign'}
	(* 3D Geometry Line *)
	FUNCTION_BLOCK Line3D EXTENDS Geometry3D


	(* Internal method *)
	METHOD FB_init : BOOL
	VAR_INPUT
		(*  if TRUE, the retain variables are initialized (warm start / cold start) *)
		bInitRetains : BOOL;
		(*  if TRUE, the instance afterwards gets moved into the copy code (online change) *)
		bInCopyCode : BOOL;
	END_VAR
END_METHOD


	(* Internal method *)
	{attribute 'hide'}
	METHOD FB_exit : BOOL
	VAR_INPUT
		(*  if TRUE, the exit method is called for exiting an instance that is copied afterwards (online change). *)
		bInCopyCode : BOOL;
	END_VAR
END_METHOD


	(* Define a line by two positions. *)
	METHOD DefineByPositions
	VAR_IN_OUT
		(* 1st position on the line to define. *)
 {attribute 'GUID' := '2AB870EB-68E4-CB90-6B70-58195CE52F48'}
				position0 : Position3D;
		(* 2nd position on the line to define. *)
 {attribute 'GUID' := '2AB870EB-68E4-CB90-6B70-58195CE52F48'}
				position1 : Position3D;
	END_VAR
END_METHOD


	(* Define a line by a position on the line and its direction. *)
	METHOD DefineByDirection
	VAR_IN_OUT
		(* Position on the line. *)
 {attribute 'GUID' := '2AB870EB-68E4-CB90-6B70-58195CE52F48'}
				position : Position3D;
		(* Direction of the line. *)
 {attribute 'GUID' := 'F5C610D1-97C6-C19E-7CED-E3534BCC46DA'}
				direction : Tangent3D;
	END_VAR
END_METHOD


	(* Set the direction of the line. *)
	METHOD SetDirection
	VAR_IN_OUT
		(* The direction to set. *)
 {attribute 'GUID' := 'F5C610D1-97C6-C19E-7CED-E3534BCC46DA'}
				direction : Tangent3D;
	END_VAR
END_METHOD


	(* Get the direction of the line. *)
	METHOD GetDirection
	VAR_IN_OUT
		(* The current direction of the line. *)
 {attribute 'GUID' := 'F5C610D1-97C6-C19E-7CED-E3534BCC46DA'}
				direction : Tangent3D;
	END_VAR
END_METHOD


	(* Get a position on the line at a specific arclength value. *)
	METHOD GetPositionAt
	VAR_INPUT
		(* Arc length value where the position is evaluated. *)
		arcLength : LREAL;
	END_VAR
	VAR_IN_OUT
		(* The position at the specified arc parameter. *)
 {attribute 'GUID' := '0AD402BA-F9BA-C1DC-7787-46186BA3F7DD'}
				position : PositionSE3;
	END_VAR
END_METHOD

END_FUNCTION_BLOCK

// POUs/Shapes/Geometry3D/1D/Circle3D

	{attribute 'c++_compatible'}
	{attribute 'external_name' := 'Circle3D_GUID_29F49B27_AAE9_CC9C_6518_224DE67B611D'}
	{attribute 'TcIecLibraryType'}
	{attribute 'no_explicit_call' :='do not call this POU directly'}
	{attribute 'no_assign'}
	FUNCTION_BLOCK Circle3D EXTENDS Geometry3D


	(* Internal method *)
	METHOD FB_init : BOOL
	VAR_INPUT
		(*  if TRUE, the retain variables are initialized (warm start / cold start) *)
		bInitRetains : BOOL;
		(*  if TRUE, the instance afterwards gets moved into the copy code (online change) *)
		bInCopyCode : BOOL;
	END_VAR
END_METHOD


	(* Internal method *)
	{attribute 'hide'}
	METHOD FB_exit : BOOL
	VAR_INPUT
		(*  if TRUE, the exit method is called for exiting an instance that is copied afterwards (online change). *)
		bInCopyCode : BOOL;
	END_VAR
END_METHOD


	(* Set the normal vector of the circle. *)
	METHOD SetNormal
	VAR_IN_OUT
		(* Normal vector to set. *)
 {attribute 'GUID' := 'F5C610D1-97C6-C19E-7CED-E3534BCC46DA'}
				normal : Tangent3D;
	END_VAR
END_METHOD


	(* Get the length of the circle. *)
	METHOD GetLength : LREAL
END_METHOD


	(* Get the normal vector of the circle. *)
	METHOD GetNormal
	VAR
		(* The current normal vector of the circle. *)
 {attribute 'GUID' := 'F5C610D1-97C6-C19E-7CED-E3534BCC46DA'}
				normal : Tangent3D;
	END_VAR
END_METHOD


	(* Get a position on the circle at a specific arclength value. *)
	METHOD GetPositionAt
	VAR_INPUT
		(* Arc length value where the position is evaluated. *)
		arcLength : LREAL;
	END_VAR
	VAR_IN_OUT
		(* The position at the specified arc parameter. *)
 {attribute 'GUID' := '0AD402BA-F9BA-C1DC-7787-46186BA3F7DD'}
				position : PositionSE3;
	END_VAR
END_METHOD


	PROPERTY radius : LREAL
SET
END_SET
GET
END_GET
END_PROPERTY

END_FUNCTION_BLOCK

// POUs/Shapes/Geometry3D/2D/Plane3D

	{attribute 'c++_compatible'}
	{attribute 'external_name' := 'Plane3D_GUID_D8C47956_A364_C74D_4E06_7A3DCBC43408'}
	{attribute 'TcIecLibraryType'}
	{attribute 'no_explicit_call' :='do not call this POU directly'}
	{attribute 'no_assign'}
	FUNCTION_BLOCK Plane3D EXTENDS Geometry3D


	(* Internal method *)
	METHOD FB_init : BOOL
	VAR_INPUT
		(*  if TRUE, the retain variables are initialized (warm start / cold start) *)
		bInitRetains : BOOL;
		(*  if TRUE, the instance afterwards gets moved into the copy code (online change) *)
		bInCopyCode : BOOL;
	END_VAR
END_METHOD


	(* Internal method *)
	{attribute 'hide'}
	METHOD FB_exit : BOOL
	VAR_INPUT
		(*  if TRUE, the exit method is called for exiting an instance that is copied afterwards (online change). *)
		bInCopyCode : BOOL;
	END_VAR
END_METHOD


	(* Set the normal of the plane. *)
	METHOD SetNormal
	VAR_IN_OUT
		(* The normal vector to set. *)
 {attribute 'GUID' := 'F5C610D1-97C6-C19E-7CED-E3534BCC46DA'}
				normal : Tangent3D;
	END_VAR
END_METHOD


	(* Get the normal vector of the plane. *)
	METHOD GetNormal
	VAR
		(* The current normal vector of the plane. *)
 {attribute 'GUID' := 'F5C610D1-97C6-C19E-7CED-E3534BCC46DA'}
				normal : Tangent3D;
	END_VAR
END_METHOD

END_FUNCTION_BLOCK

// POUs/Shapes/Geometry3D/2D/Disc3D

	{attribute 'c++_compatible'}
	{attribute 'external_name' := 'Disc3D_GUID_427A9789_3187_CB59_44A8_2D8FAAC25A4A'}
	{attribute 'TcIecLibraryType'}
	{attribute 'no_explicit_call' :='do not call this POU directly'}
	{attribute 'no_assign'}
	FUNCTION_BLOCK Disc3D EXTENDS Geometry3D


	(* Internal method *)
	METHOD FB_init : BOOL
	VAR_INPUT
		(*  if TRUE, the retain variables are initialized (warm start / cold start) *)
		bInitRetains : BOOL;
		(*  if TRUE, the instance afterwards gets moved into the copy code (online change) *)
		bInCopyCode : BOOL;
	END_VAR
END_METHOD


	(* Internal method *)
	{attribute 'hide'}
	METHOD FB_exit : BOOL
	VAR_INPUT
		(*  if TRUE, the exit method is called for exiting an instance that is copied afterwards (online change). *)
		bInCopyCode : BOOL;
	END_VAR
END_METHOD


	(* Set the normal vector of the disc. *)
	METHOD SetNormal
	VAR_IN_OUT
		(* The normal to set. *)
 {attribute 'GUID' := 'F5C610D1-97C6-C19E-7CED-E3534BCC46DA'}
				normal : Tangent3D;
	END_VAR
END_METHOD


	(* Get the normal vector of the disc. *)
	METHOD GetNormal
	VAR
		(* The current normal vector of the disc. *)
 {attribute 'GUID' := 'F5C610D1-97C6-C19E-7CED-E3534BCC46DA'}
				normal : Tangent3D;
	END_VAR
END_METHOD


	(* Get the area of the disc. *)
	METHOD GetArea : LREAL
END_METHOD


	PROPERTY radius : LREAL
SET
END_SET
GET
END_GET
END_PROPERTY

END_FUNCTION_BLOCK

// POUs/Shapes/Geometry3D/2D/Rectangle3D

	{attribute 'c++_compatible'}
	{attribute 'external_name' := 'Rectangle3D_GUID_10F404C4_E301_C3CE_66AE_823B6045FA74'}
	{attribute 'TcIecLibraryType'}
	{attribute 'no_explicit_call' :='do not call this POU directly'}
	{attribute 'no_assign'}
	FUNCTION_BLOCK Rectangle3D EXTENDS Geometry3D


	(* Internal method *)
	METHOD FB_init : BOOL
	VAR_INPUT
		(*  if TRUE, the retain variables are initialized (warm start / cold start) *)
		bInitRetains : BOOL;
		(*  if TRUE, the instance afterwards gets moved into the copy code (online change) *)
		bInCopyCode : BOOL;
	END_VAR
END_METHOD


	(* Internal method *)
	{attribute 'hide'}
	METHOD FB_exit : BOOL
	VAR_INPUT
		(*  if TRUE, the exit method is called for exiting an instance that is copied afterwards (online change). *)
		bInCopyCode : BOOL;
	END_VAR
END_METHOD


	(* Set the dimensions of the rectangle. *)
	METHOD SetDimensions
	VAR_INPUT
		(* The width of the rectangle to set. *)
		width : LREAL;
		(* The height of the rectangle to set. *)
		height : LREAL;
	END_VAR
END_METHOD


	(* Get the area of the rectangle. *)
	METHOD GetArea : LREAL
END_METHOD


	PROPERTY width : LREAL
SET
END_SET
GET
END_GET
END_PROPERTY


	PROPERTY height : LREAL
SET
END_SET
GET
END_GET
END_PROPERTY

END_FUNCTION_BLOCK

// POUs/Shapes/Geometry3D/3D/Sphere3D

	{attribute 'c++_compatible'}
	{attribute 'external_name' := 'Sphere3D_GUID_EA1C09E9_BD9B_C6DF_75C8_FCB2746D9A16'}
	{attribute 'TcIecLibraryType'}
	{attribute 'no_explicit_call' :='do not call this POU directly'}
	{attribute 'no_assign'}
	FUNCTION_BLOCK Sphere3D EXTENDS Geometry3D


	(* Internal method *)
	METHOD FB_init : BOOL
	VAR_INPUT
		(*  if TRUE, the retain variables are initialized (warm start / cold start) *)
		bInitRetains : BOOL;
		(*  if TRUE, the instance afterwards gets moved into the copy code (online change) *)
		bInCopyCode : BOOL;
	END_VAR
END_METHOD


	(* Internal method *)
	{attribute 'hide'}
	METHOD FB_exit : BOOL
	VAR_INPUT
		(*  if TRUE, the exit method is called for exiting an instance that is copied afterwards (online change). *)
		bInCopyCode : BOOL;
	END_VAR
END_METHOD


	(* Get the volume of the sphere. *)
	METHOD GetVolume : LREAL
END_METHOD


	PROPERTY radius : LREAL
SET
END_SET
GET
END_GET
END_PROPERTY

END_FUNCTION_BLOCK

// POUs/Shapes/Geometry3D/3D/Cuboid3D

	{attribute 'c++_compatible'}
	{attribute 'external_name' := 'Cuboid3D_GUID_18069D6A_C874_C0E8_4FEF_226945B11EBE'}
	{attribute 'TcIecLibraryType'}
	{attribute 'no_explicit_call' :='do not call this POU directly'}
	{attribute 'no_assign'}
	FUNCTION_BLOCK Cuboid3D EXTENDS Geometry3D


	(* Internal method *)
	METHOD FB_init : BOOL
	VAR_INPUT
		(* if TRUE, the retain variables are initialized (warm start / cold start) *)
		bInitRetains : BOOL;
		(* if TRUE, the instance afterwards gets moved into the copy code (online change) *)
		bInCopyCode : BOOL;
	END_VAR
END_METHOD


	(* Internal method *)
	{attribute 'hide'}
	METHOD FB_exit : BOOL
	VAR_INPUT
		(* if TRUE, the exit method is called for exiting an instance that is copied afterwards (online change). *)
		bInCopyCode : BOOL;
	END_VAR
END_METHOD


	(* Set the dimensions of the cuboid. *)
	METHOD SetDimensions
	VAR_INPUT
		(* local x-component *)
		length : LREAL;
		(* local y-component *)
		width : LREAL;
		(* local z-component *)
		height : LREAL;
	END_VAR
END_METHOD


	(* Get the volume of the cuboid. *)
	METHOD GetVolume : LREAL
END_METHOD


	PROPERTY length : LREAL
SET
END_SET
GET
END_GET
END_PROPERTY


	PROPERTY width : LREAL
SET
END_SET
GET
END_GET
END_PROPERTY


	PROPERTY height : LREAL
SET
END_SET
GET
END_GET
END_PROPERTY

END_FUNCTION_BLOCK

// POUs/Shapes/Geometry3D/3D/Cylinder3D

	{attribute 'c++_compatible'}
	{attribute 'external_name' := 'Cylinder3D_GUID_7C98C750_EF5C_C80A_51BC_9CA264194E19'}
	{attribute 'TcIecLibraryType'}
	{attribute 'no_explicit_call' :='do not call this POU directly'}
	{attribute 'no_assign'}
	FUNCTION_BLOCK Cylinder3D EXTENDS Geometry3D


	(* Internal method *)
	METHOD FB_init : BOOL
	VAR_INPUT
		(* if TRUE, the retain variables are initialized (warm start / cold start) *)
		bInitRetains : BOOL;
		(* if TRUE, the instance afterwards gets moved into the copy code (online change) *)
		bInCopyCode : BOOL;
	END_VAR
END_METHOD


	(* Internal method *)
	{attribute 'hide'}
	METHOD FB_exit : BOOL
	VAR_INPUT
		(* if TRUE, the exit method is called for exiting an instance that is copied afterwards (online change). *)
		bInCopyCode : BOOL;
	END_VAR
END_METHOD


	(* Set the dimensions of the cylinder. *)
	METHOD SetDimensions
	VAR_INPUT
		(* The radius to set. *)
		radius : LREAL;
		(* The height to set. *)
		height : LREAL;
	END_VAR
END_METHOD


	(* Get the volume of the cylinder. *)
	METHOD GetVolume : LREAL
END_METHOD


	PROPERTY radius : LREAL
SET
END_SET
GET
END_GET
END_PROPERTY


	PROPERTY height : LREAL
SET
END_SET
GET
END_GET
END_PROPERTY

END_FUNCTION_BLOCK
